(* Logix 5000 project; controller DIMTER vendor 1 type 14 code 77 rev 15.4; software revision 15.01; part 2 of 4 *)
(* tags used below, declared in another part *)
   F : BOOL[2016];   // Flags
   T : TIMER[100];   // Timers
   A123 : ALIAS FOR Local:4:O.Data.3;   // O:4.0/3 A12.3 Reset Buffer
   A142 : ALIAS FOR Local:5:O.Data.2;   // O:5.0/2 A142 Raise Rake 1
   A143 : ALIAS FOR Local:5:O.Data.3;   // O:5.0/3 A143 Brake Cross Conveyor Front of Saw 1
   A144 : ALIAS FOR Local:5:O.Data.4;   // O:5.0/4 A144 Cross Feed 1 Fast Fwd
   A145 : ALIAS FOR Local:5:O.Data.5;   // O:5.0/5 A145 Cross Feed 1 Slow Fwd
   A146 : ALIAS FOR Local:5:O.Data.6;   // O:5.0/6 A146 Cross Feed 1 Fast Rev
   A152 : ALIAS FOR Local:5:O.Data.10;   // O:5.0/10 A15.2 Forward Rotation Rollcase 1
   A156 : ALIAS FOR Local:5:O.Data.14;   // O:5.0/14 A156 Forward Rotation Rollcase 2
   A162 : ALIAS FOR Local:6:O.Data.2;   // O:6.0/2 A16.2 Rake 2
   A163 : ALIAS FOR Local:6:O.Data.3;   // O:6.0/3 A16.3 Brake Cross Conveyor Front of Saw 2
   A164 : ALIAS FOR Local:6:O.Data.4;   // O:6.0/4 A16.4 Cross Feed 2 Fast Fwd
   A165 : ALIAS FOR Local:6:O.Data.5;   // O:6.0/5 A16.5 Cross Feed 2 Slow Fwd
   A166 : ALIAS FOR Local:6:O.Data.6;   // O:6.0/6 A16.6 Cross Feed 2 Fast Rev
   A170 : ALIAS FOR Local:6:O.Data.8;   // O:6.0/8 A17.0 Infeed Measuring Slot Weinig Release Workpiece to Demand
   A171 : ALIAS FOR Local:6:O.Data.9;   // O:6.0/9 A17.1 Conveyor Measuring Slot Weinig Feed to Switch On
   A184 : ALIAS FOR Local:7:O.Data.4;   // O:7.0/4 A18.4 Waste Belt Conveyor 1
   A185 : ALIAS FOR Local:7:O.Data.5;   // O:7.0/5 A18.5 Waste Belt Conveyor 2
   A186 : ALIAS FOR Local:7:O.Data.6;   // O:7.0/6 A18.6 Cross Belt 1
   A187 : ALIAS FOR Local:7:O.Data.7;   // O:7.0/7 A18.7 Cross Belt 2
   E01 : ALIAS FOR Local:1:I.Data.1;   // I:1.0/1 E0.1 Saw Hood 1 Closed
   E02 : ALIAS FOR Local:1:I.Data.2;   // I:1.0/2 E0.2 Saw Motor 1 On
   E05 : ALIAS FOR Local:1:I.Data.5;   // I:1.0/5 E0.5 Failure Chain Ejector
   E06 : ALIAS FOR Local:1:I.Data.6;   // I:1.0/6 E0.6 Failure Conveyor in Front of Saw 1
   E07 : ALIAS FOR Local:1:I.Data.7;   // I:1.0/7 E0.7 Failure Conveyor in Front of Saw 2
   E10 : ALIAS FOR Local:1:I.Data.8;   // I:1.0/8 E1.0 Failure Weinig Conveyor
   E100 : ALIAS FOR Local:3:I.Data.16;   // I:3.1/0 E10.0 Sorting Ejector Sorting 1
   E101 : ALIAS FOR Local:3:I.Data.17;   // I:3.1/1 E10.1 Sorting Ejector 2 Sorting 1
   E102 : ALIAS FOR Local:3:I.Data.18;   // I:3.1/2 E10.2 Sorting Ejector 3 Sorting 1
   E103 : ALIAS FOR Local:3:I.Data.19;   // I:3.1/3 E10.3 Sorting Ejector 1 Sorting 2
   E104 : ALIAS FOR Local:3:I.Data.20;   // I:3.1/4 E10.4 Sorting Ejector 2 Sorting 2
   E105 : ALIAS FOR Local:3:I.Data.21;   // I:3.1/5 E10.5 Sorting Ejector 3 Sorting 2
   E106 : ALIAS FOR Local:3:I.Data.22;   // I:3.1/6 E10.6 Cross Belt 1 Cyclewise Continuous Running
   E107 : ALIAS FOR Local:3:I.Data.23;   // I:3.1/7 E10.7 ???
   E11 : ALIAS FOR Local:1:I.Data.9;   // I:1.0/9 E1.1 Saw Hood 2 Closed
   E110 : ALIAS FOR Local:3:I.Data.24;   // I:3.1/8 E11.0 Cross Belt 1 Footswitch (Removed)
   E111 : ALIAS FOR Local:3:I.Data.25;   // I:3.1/9 E11.1 Cross Belt 2 Cyclewise Continuous Running
   E112 : ALIAS FOR Local:3:I.Data.26;   // I:3.1/10 E11.2 ???
   E113 : ALIAS FOR Local:3:I.Data.27;   // I:3.1/11 E11.3 Cross Belt 2 Footswitch (Removed)
   E114 : ALIAS FOR Local:3:I.Data.28;   // I:3.1/12 E11.4 Transfer Station On
   E115 : ALIAS FOR Local:3:I.Data.29;   // I:3.1/13 E11.5 Cross Feed Manual Fwd-Rev
   E116 : ALIAS FOR Local:3:I.Data.30;   // I:3.1/14 E11.6 ???
   E12 : ALIAS FOR Local:1:I.Data.10;   // I:1.0/10 E1.2 Saw Motor 2 On
   E20 : ALIAS FOR Local:1:I.Data.16;   // I:1.1/0 E2.0 Protection Hood Measuring System
   E27 : ALIAS FOR Local:1:I.Data.23;   // I:1.1/7 E2.7 Reset Safety Barrier at Transfer Station
   E41 : ALIAS FOR Local:2:I.Data.1;   // I:2.0/1 E4.1 Cross Feed 1 Manual Fwd - Rev
   E42 : ALIAS FOR Local:2:I.Data.2;   // I:2.0/2 E4.2 Cross Feed 1 Manual Fwd - Rev
   E44 : ALIAS FOR Local:2:I.Data.4;   // I:2.0/4 E4.4 Waste Conveyor Belt On
   E45 : ALIAS FOR Local:2:I.Data.5;   // I:2.0/5 E4.5 Transfer Station in Front of Saw On
   E51 : ALIAS FOR Local:2:I.Data.9;   // I:2.0/9 E5.1 Cross Feed 2 Manual Fwd - Rev
   E52 : ALIAS FOR Local:2:I.Data.10;   // I:2.0/10 E5.2 Cross Feed 2 Manual Fwd - Rev
   E54 : ALIAS FOR Local:2:I.Data.12;   // I:2.0/12 E5.4 Measuring Station On
   E57 : ALIAS FOR Local:2:I.Data.15;   // I:2.0/15 E5.7 Conveyor Measuring Station Manual
   E67 : ALIAS FOR Local:2:I.Data.23;   // I:2.1/7 E6.7 PE Cross Feed 1 Waiting Position
   E72 : ALIAS FOR Local:2:I.Data.26;   // I:2.1/10 E7.2 Stop Rollcase 1
   E73 : ALIAS FOR Local:2:I.Data.27;   // I:2.1/11 E7.3 Cross Feed 1 Down
   E74 : ALIAS FOR Local:2:I.Data.28;   // I:2.1/12 E7.4 Cross Feed 1 Up
   E75 : ALIAS FOR Local:2:I.Data.29;   // I:2.1/13 E7.5 Cross Feed 1 Initial Position
   E76 : ALIAS FOR Local:2:I.Data.30;   // I:2.1/14 E7.6 PE Cross Feed 1 Slow Fwd
   E77 : ALIAS FOR Local:2:I.Data.31;   // I:2.1/15 E7.7 Cross Feed 1 at Front
   E87 : ALIAS FOR Local:3:I.Data.7;   // I:3.0/7 E8.7 PE Cross Feed 2 Waiting Position
   E92 : ALIAS FOR Local:3:I.Data.10;   // I:3.0/10 E9.2 Stop Rollcase 2
   E93 : ALIAS FOR Local:3:I.Data.11;   // I:3.0/11 E9.3 Cross Feed 2 Down
   E94 : ALIAS FOR Local:3:I.Data.12;   // I:3.0/12 E9.4 Cross Feed 2 Up
   E95 : ALIAS FOR Local:3:I.Data.13;   // I:3.0/13 E9.5 Cross Feed 2 Home Position
   E96 : ALIAS FOR Local:3:I.Data.14;   // I:3.0/14 E9.6 PE Cross Feed 2 Slow Fwd
   E97 : ALIAS FOR Local:3:I.Data.15;   // I:3.0/15 E9.7 Cross Feed 2 at Front
(* MainProgram, continued *)

ROUTINE Conveyors   (* ladder *)
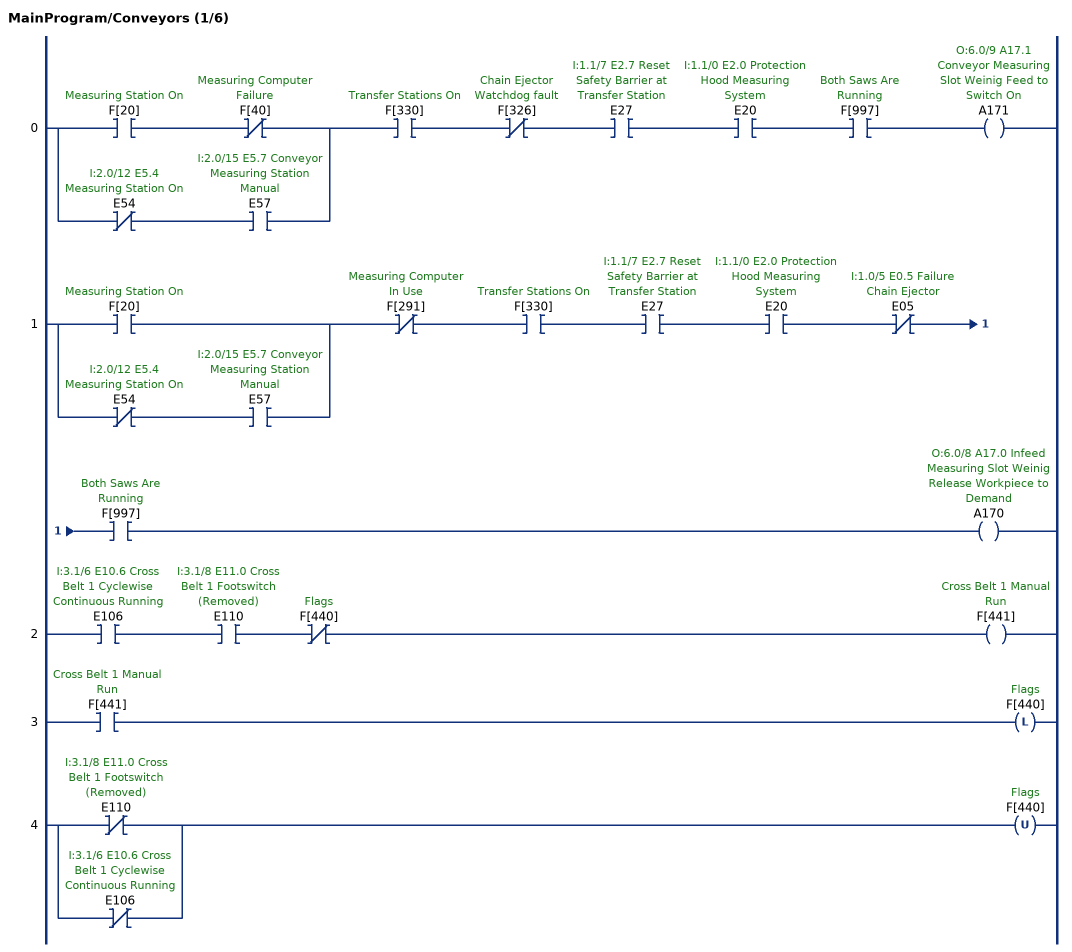
   0: [XIC(F[20]) XIO(F[40]) ,XIO(E54) XIC(E57) ]XIC(F[330])XIO(F[326])XIC(E27)XIC(E20)XIC(F[997])OTE(A171);
   1: [XIC(F[20]) ,XIO(E54) XIC(E57) ]XIO(F[291])XIC(F[330])XIC(E27)XIC(E20)XIO(E05)XIC(F[997])OTE(A170);
   2: XIC(E106)XIC(E110)XIO(F[440])OTE(F[441]);
   3: XIC(F[441])OTL(F[440]);
   4: [XIO(E110) ,XIO(E106) ]OTU(F[440]);
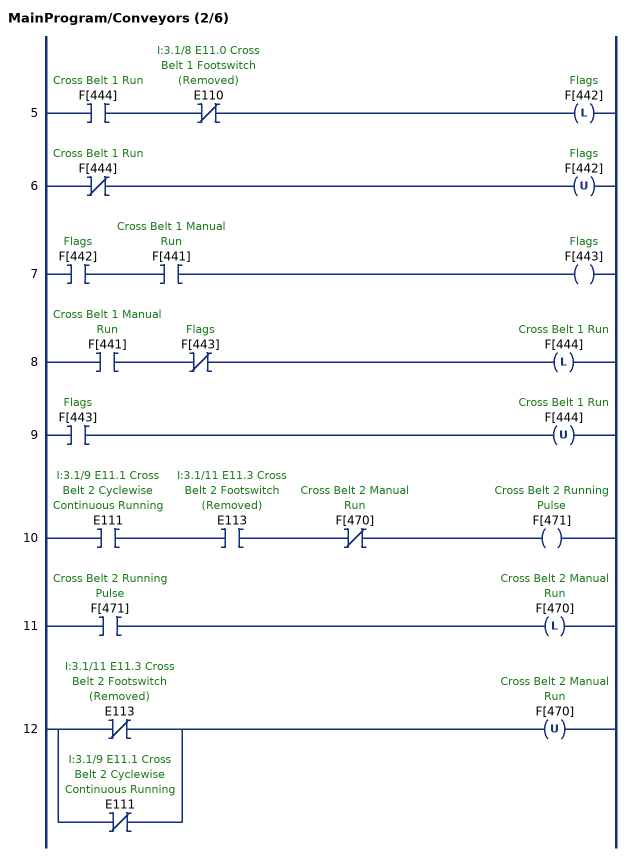
   5: XIC(F[444])XIO(E110)OTL(F[442]);
   6: XIO(F[444])OTU(F[442]);
   7: XIC(F[442])XIC(F[441])OTE(F[443]);
   8: XIC(F[441])XIO(F[443])OTL(F[444]);
   9: XIC(F[443])OTU(F[444]);
   10: XIC(E111)XIC(E113)XIO(F[470])OTE(F[471]);
   11: XIC(F[471])OTL(F[470]);
   12: [XIO(E113) ,XIO(E111) ]OTU(F[470]);
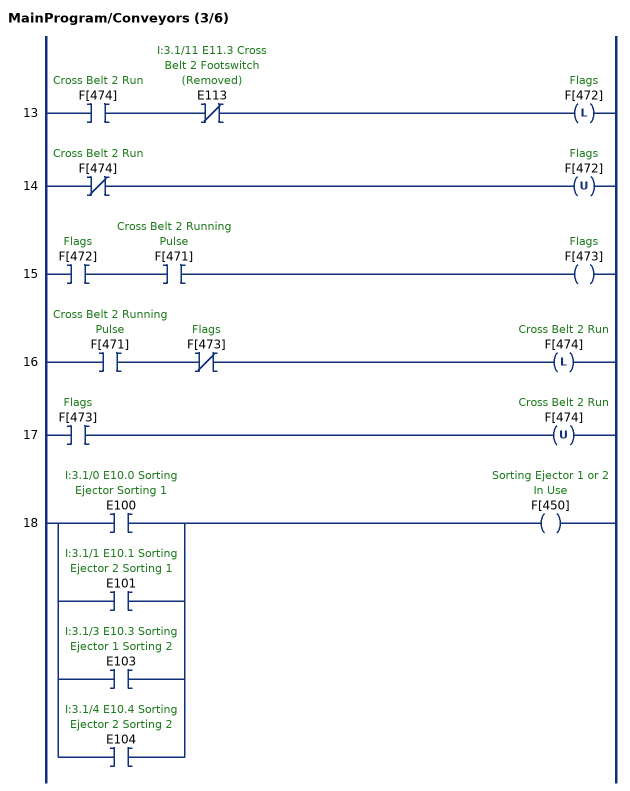
   13: XIC(F[474])XIO(E113)OTL(F[472]);
   14: XIO(F[474])OTU(F[472]);
   15: XIC(F[472])XIC(F[471])OTE(F[473]);
   16: XIC(F[471])XIO(F[473])OTL(F[474]);
   17: XIC(F[473])OTU(F[474]);
   18: [XIC(E100) ,XIC(E101) ,XIC(E103) ,XIC(E104) ]OTE(F[450]);
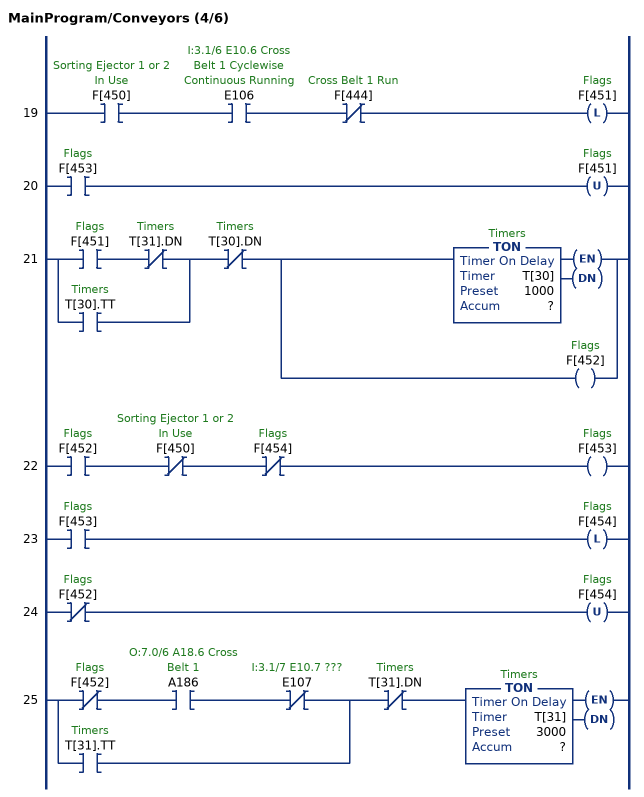
   19: XIC(F[450])XIC(E106)XIO(F[444])OTL(F[451]);
   20: XIC(F[453])OTU(F[451]);
   21: [XIC(F[451]) XIO(T[31].DN) ,XIC(T[30].TT) ]XIO(T[30].DN)[TON(T[30],?,?) ,OTE(F[452]) ];
   22: XIC(F[452])XIO(F[450])XIO(F[454])OTE(F[453]);
   23: XIC(F[453])OTL(F[454]);
   24: XIO(F[452])OTU(F[454]);
   25: [XIO(F[452]) XIC(A186) XIO(E107) ,XIC(T[31].TT) ]XIO(T[31].DN)TON(T[31],?,?);
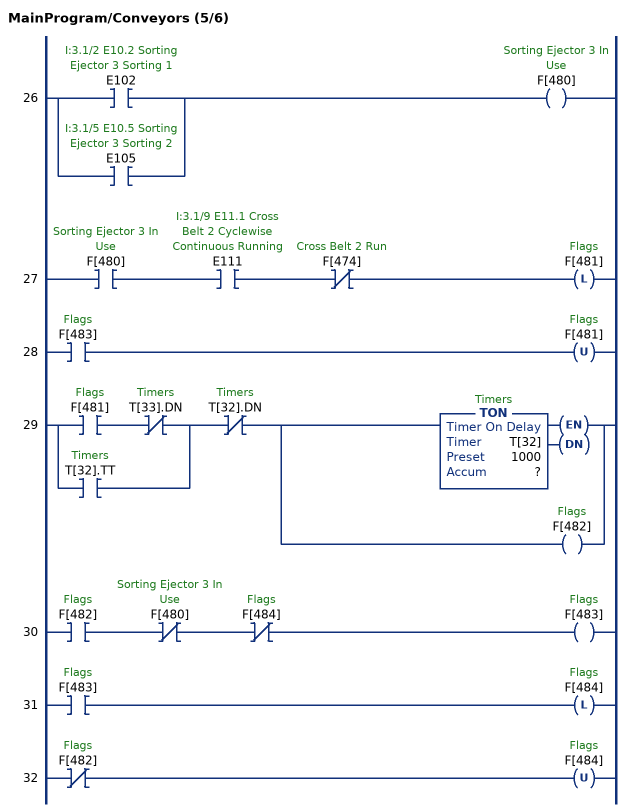
   26: [XIC(E102) ,XIC(E105) ]OTE(F[480]);
   27: XIC(F[480])XIC(E111)XIO(F[474])OTL(F[481]);
   28: XIC(F[483])OTU(F[481]);
   29: [XIC(F[481]) XIO(T[33].DN) ,XIC(T[32].TT) ]XIO(T[32].DN)[TON(T[32],?,?) ,OTE(F[482]) ];
   30: XIC(F[482])XIO(F[480])XIO(F[484])OTE(F[483]);
   31: XIC(F[483])OTL(F[484]);
   32: XIO(F[482])OTU(F[484]);
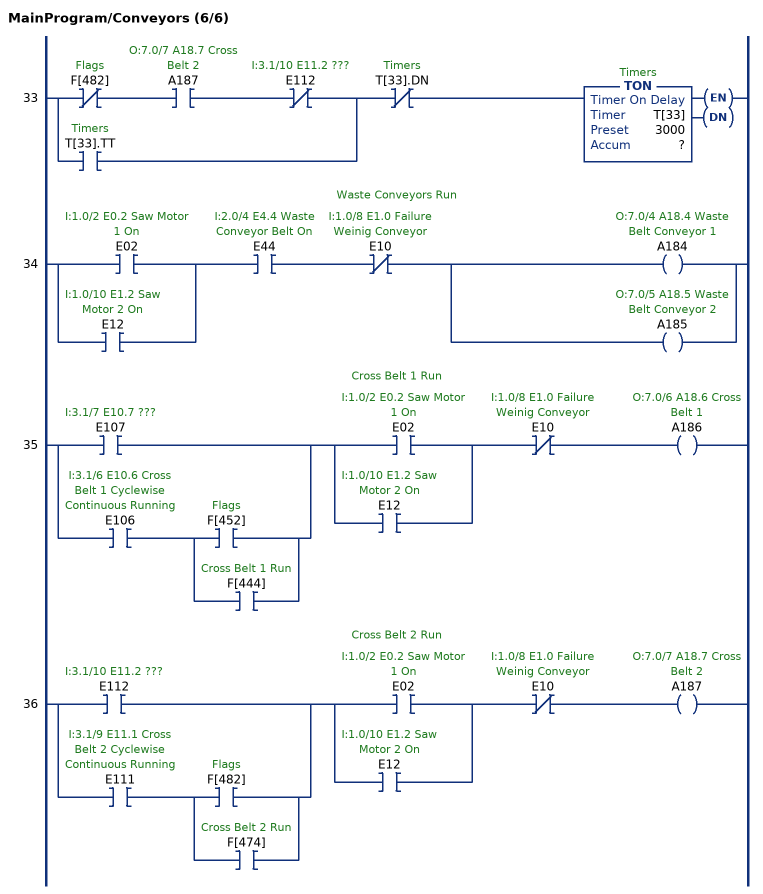
   33: [XIO(F[482]) XIC(A187) XIO(E112) ,XIC(T[33].TT) ]XIO(T[33].DN)TON(T[33],?,?);
   // Waste Conveyors Run
   34: [XIC(E02) ,XIC(E12) ]XIC(E44)XIO(E10)[OTE(A184) ,OTE(A185) ];
   // Cross Belt 1 Run
   35: [XIC(E107) ,XIC(E106) [XIC(F[452]) ,XIC(F[444]) ] ][XIC(E02) ,XIC(E12) ]XIO(E10)OTE(A186);
   // Cross Belt 2 Run
   36: [XIC(E112) ,XIC(E111) [XIC(F[482]) ,XIC(F[474]) ] ][XIC(E02) ,XIC(E12) ]XIO(E10)OTE(A187);
END_ROUTINE

ROUTINE CrossFeeds   (* ladder *)
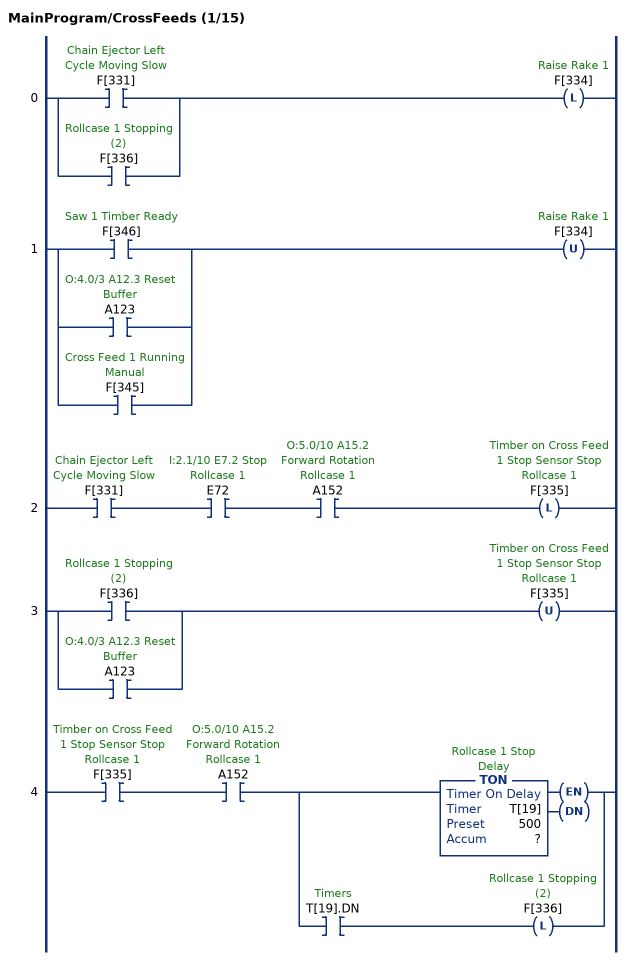
   0: [XIC(F[331]) ,XIC(F[336]) ]OTL(F[334]);
   1: [XIC(F[346]) ,XIC(A123) ,XIC(F[345]) ]OTU(F[334]);
   2: XIC(F[331])XIC(E72)XIC(A152)OTL(F[335]);
   3: [XIC(F[336]) ,XIC(A123) ]OTU(F[335]);
   4: XIC(F[335])XIC(A152)[TON(T[19],?,?) ,XIC(T[19].DN) OTL(F[336]) ];
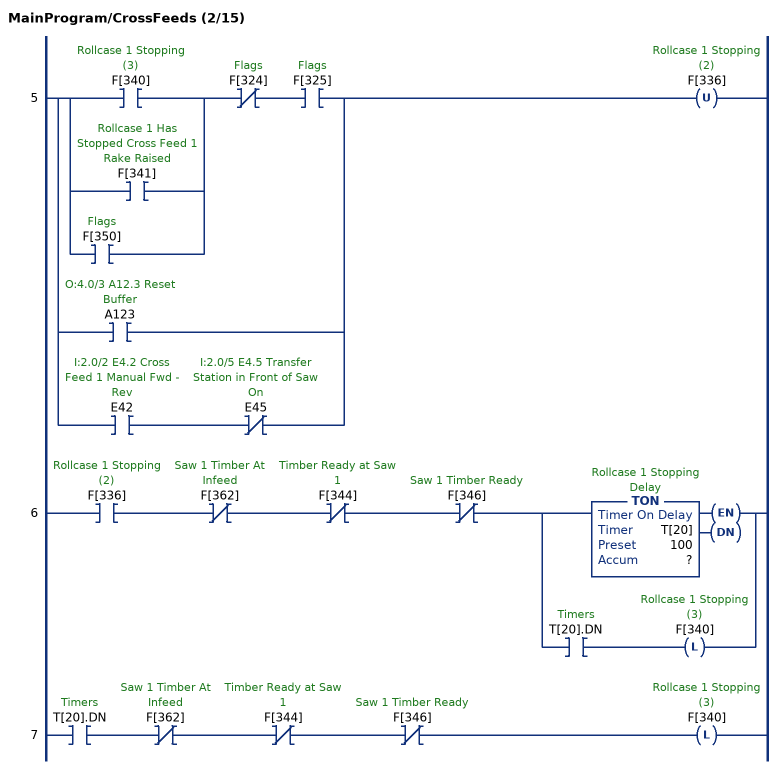
   5: [[XIC(F[340]) ,XIC(F[341]) ,XIC(F[350]) ] XIO(F[324]) XIC(F[325]) ,XIC(A123) ,XIC(E42) XIO(E45) ]OTU(F[336]);
   6: XIC(F[336])XIO(F[362])XIO(F[344])XIO(F[346])[TON(T[20],?,?) ,XIC(T[20].DN) OTL(F[340]) ];
   7: XIC(T[20].DN)XIO(F[362])XIO(F[344])XIO(F[346])OTL(F[340]);
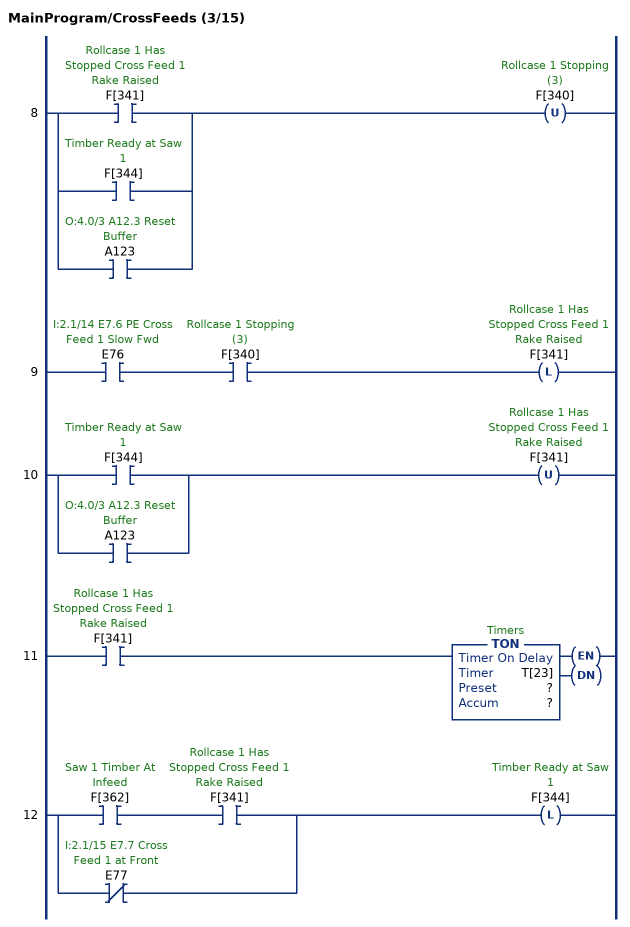
   8: [XIC(F[341]) ,XIC(F[344]) ,XIC(A123) ]OTU(F[340]);
   9: XIC(E76)XIC(F[340])OTL(F[341]);
   10: [XIC(F[344]) ,XIC(A123) ]OTU(F[341]);
   11: XIC(F[341])TON(T[23],?,?);
   12: [XIC(F[362]) XIC(F[341]) ,XIO(E77) ]OTL(F[344]);
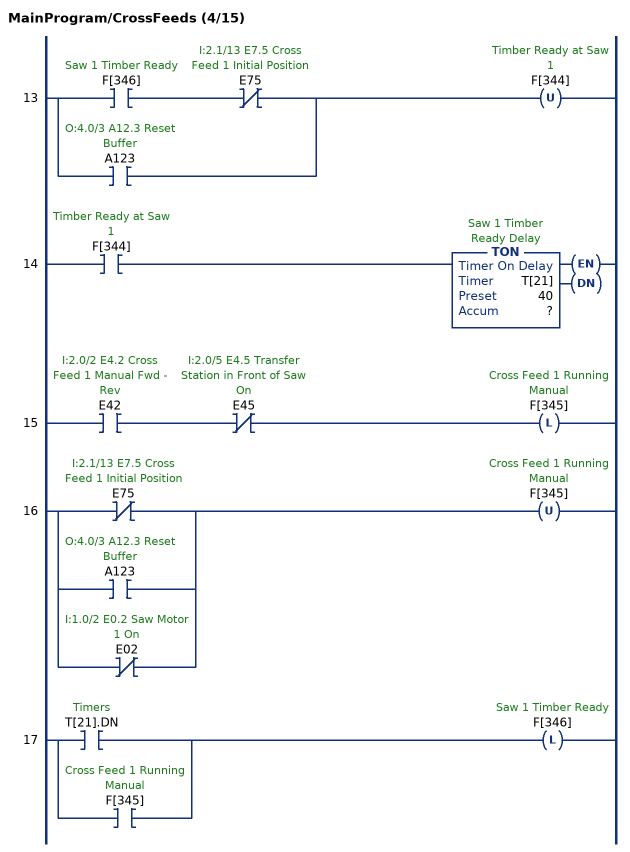
   13: [XIC(F[346]) XIO(E75) ,XIC(A123) ]OTU(F[344]);
   14: XIC(F[344])TON(T[21],?,?);
   15: XIC(E42)XIO(E45)OTL(F[345]);
   16: [XIO(E75) ,XIC(A123) ,XIO(E02) ]OTU(F[345]);
   17: [XIC(T[21].DN) ,XIC(F[345]) ]OTL(F[346]);
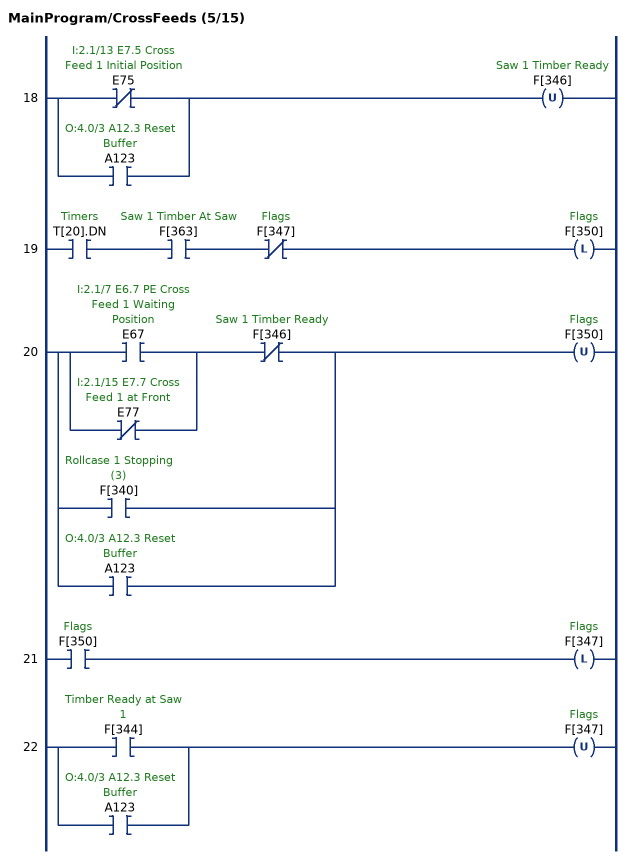
   18: [XIO(E75) ,XIC(A123) ]OTU(F[346]);
   19: XIC(T[20].DN)XIC(F[363])XIO(F[347])OTL(F[350]);
   20: [[XIC(E67) ,XIO(E77) ] XIO(F[346]) ,XIC(F[340]) ,XIC(A123) ]OTU(F[350]);
   21: XIC(F[350])OTL(F[347]);
   22: [XIC(F[344]) ,XIC(A123) ]OTU(F[347]);
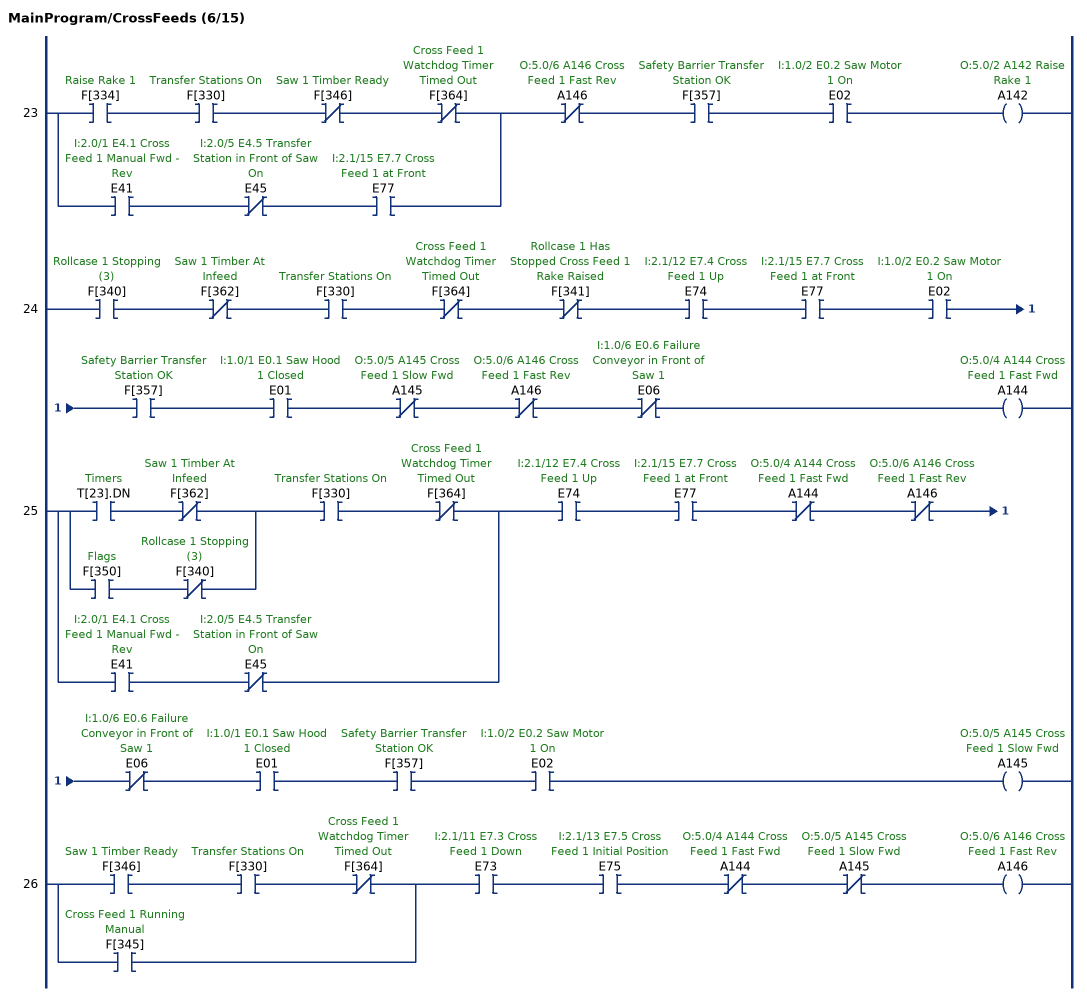
   23: [XIC(F[334]) XIC(F[330]) XIO(F[346]) XIO(F[364]) ,XIC(E41) XIO(E45) XIC(E77) ]XIO(A146)XIC(F[357])XIC(E02)OTE(A142);
   24: XIC(F[340])XIO(F[362])XIC(F[330])XIO(F[364])XIO(F[341])XIC(E74)XIC(E77)XIC(E02)XIC(F[357])XIC(E01)XIO(A145)XIO(A146)XIO(E06)OTE(A144);
   25: [[XIC(T[23].DN) XIO(F[362]) ,XIC(F[350]) XIO(F[340]) ] XIC(F[330]) XIO(F[364]) ,XIC(E41) XIO(E45) ]XIC(E74)XIC(E77)XIO(A144)XIO(A146)XIO(E06)XIC(E01)XIC(F[357])XIC(E02)OTE(A145);
   26: [XIC(F[346]) XIC(F[330]) XIO(F[364]) ,XIC(F[345]) ]XIC(E73)XIC(E75)XIO(A144)XIO(A145)OTE(A146);
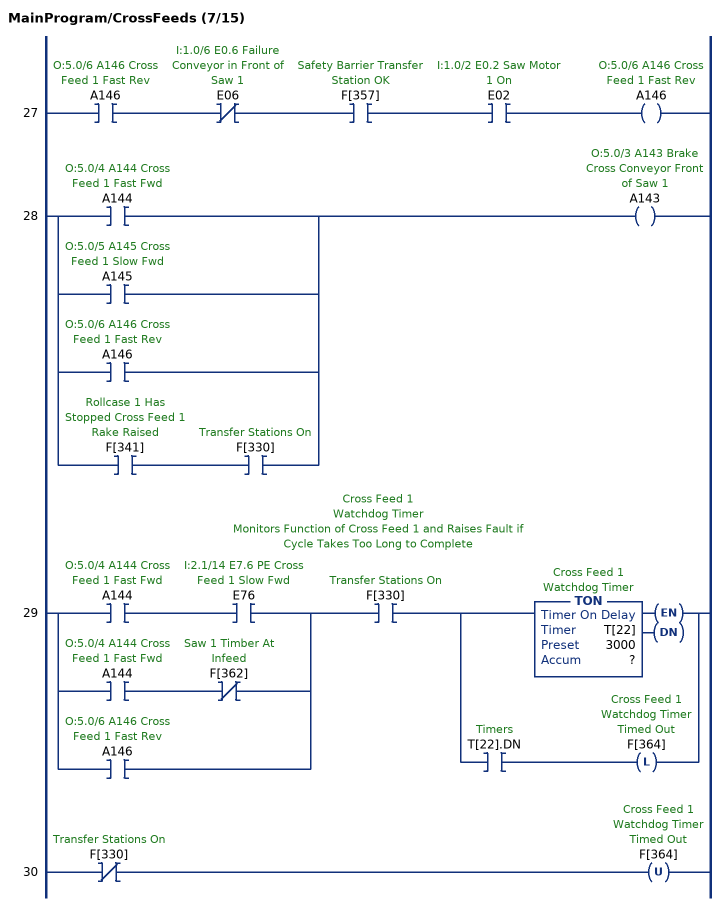
   27: XIC(A146)XIO(E06)XIC(F[357])XIC(E02)OTE(A146);
   28: [XIC(A144) ,XIC(A145) ,XIC(A146) ,XIC(F[341]) XIC(F[330]) ]OTE(A143);
   // Cross Feed 1
   // Watchdog Timer
   // Monitors Function of Cross Feed 1 and Raises Fault if
   // Cycle Takes Too Long to Complete
   29: [XIC(A144) XIC(E76) ,XIC(A144) XIO(F[362]) ,XIC(A146) ]XIC(F[330])[TON(T[22],?,?) ,XIC(T[22].DN) OTL(F[364]) ];
   30: XIO(F[330])OTU(F[364]);
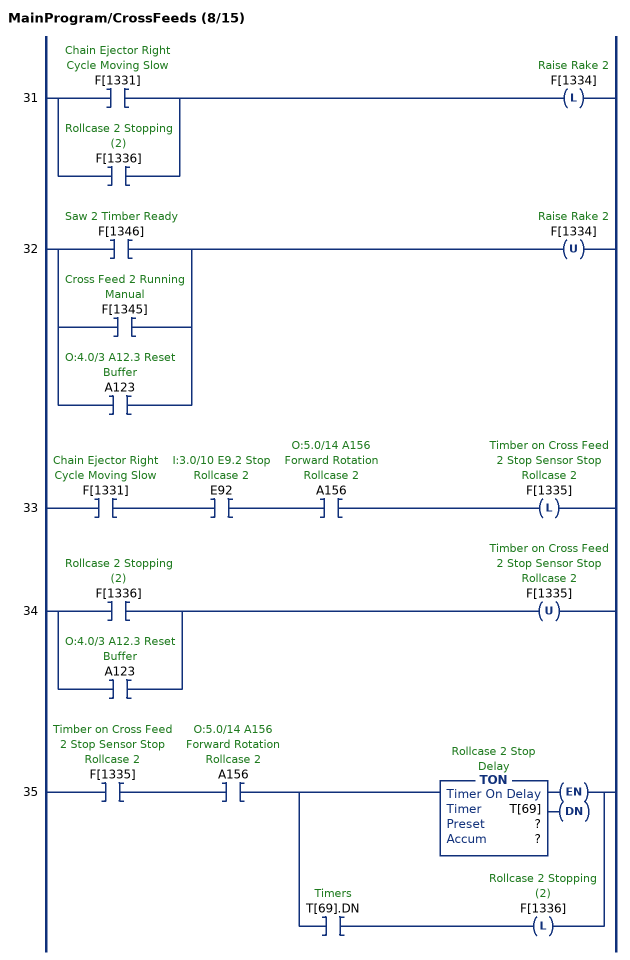
   31: [XIC(F[1331]) ,XIC(F[1336]) ]OTL(F[1334]);
   32: [XIC(F[1346]) ,XIC(F[1345]) ,XIC(A123) ]OTU(F[1334]);
   33: XIC(F[1331])XIC(E92)XIC(A156)OTL(F[1335]);
   34: [XIC(F[1336]) ,XIC(A123) ]OTU(F[1335]);
   35: XIC(F[1335])XIC(A156)[TON(T[69],?,?) ,XIC(T[69].DN) OTL(F[1336]) ];
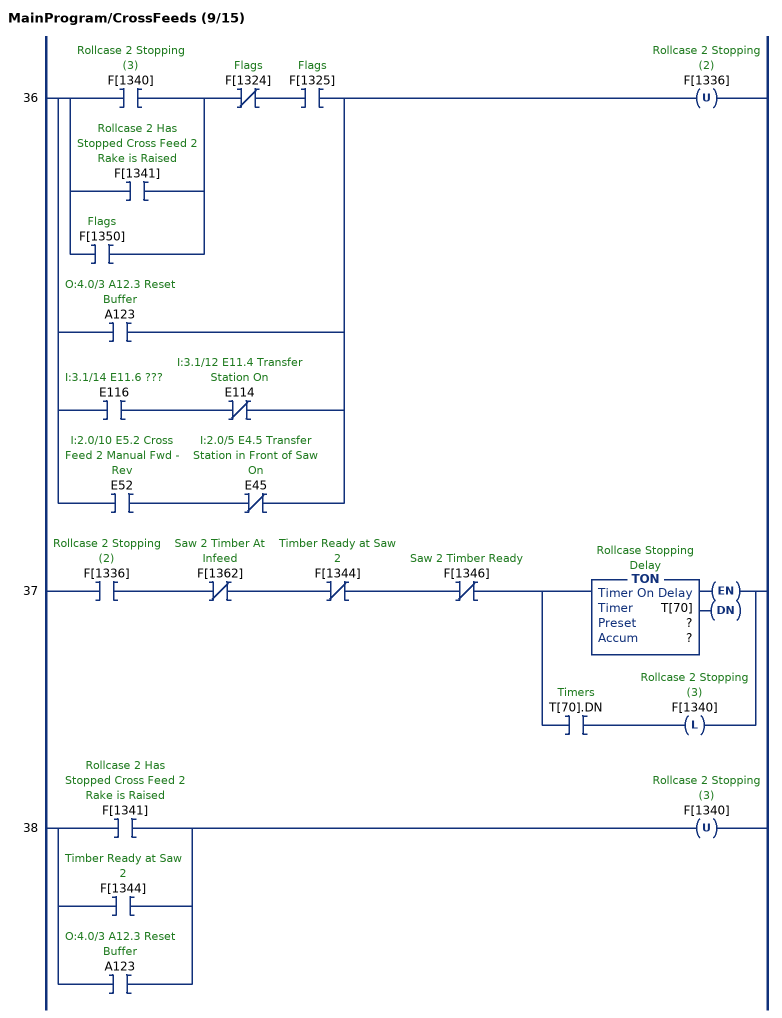
   36: [[XIC(F[1340]) ,XIC(F[1341]) ,XIC(F[1350]) ] XIO(F[1324]) XIC(F[1325]) ,XIC(A123) ,XIC(E116) XIO(E114) ,XIC(E52) XIO(E45) ]OTU(F[1336]);
   37: XIC(F[1336])XIO(F[1362])XIO(F[1344])XIO(F[1346])[TON(T[70],?,?) ,XIC(T[70].DN) OTL(F[1340]) ];
   38: [XIC(F[1341]) ,XIC(F[1344]) ,XIC(A123) ]OTU(F[1340]);
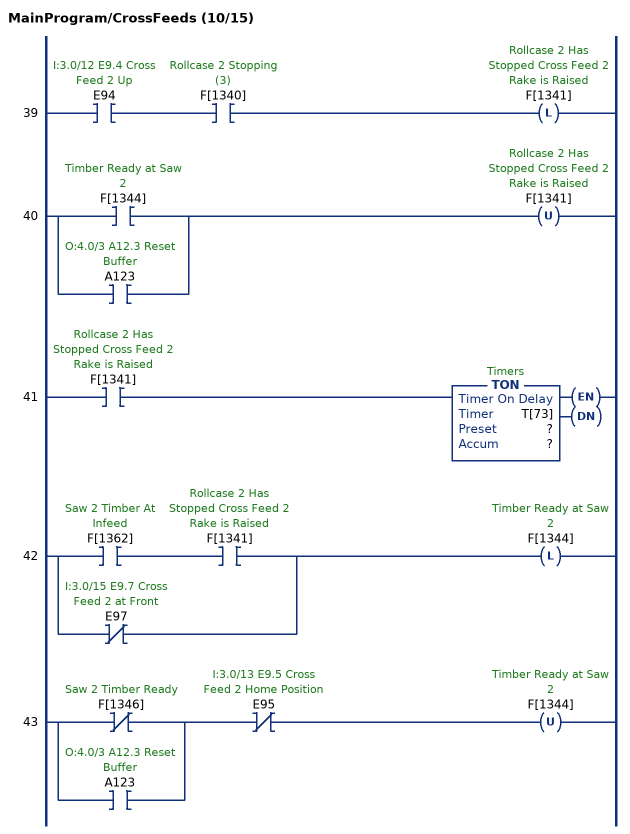
   39: XIC(E94)XIC(F[1340])OTL(F[1341]);
   40: [XIC(F[1344]) ,XIC(A123) ]OTU(F[1341]);
   41: XIC(F[1341])TON(T[73],?,?);
   42: [XIC(F[1362]) XIC(F[1341]) ,XIO(E97) ]OTL(F[1344]);
   43: [XIO(F[1346]) ,XIC(A123) ]XIO(E95)OTU(F[1344]);
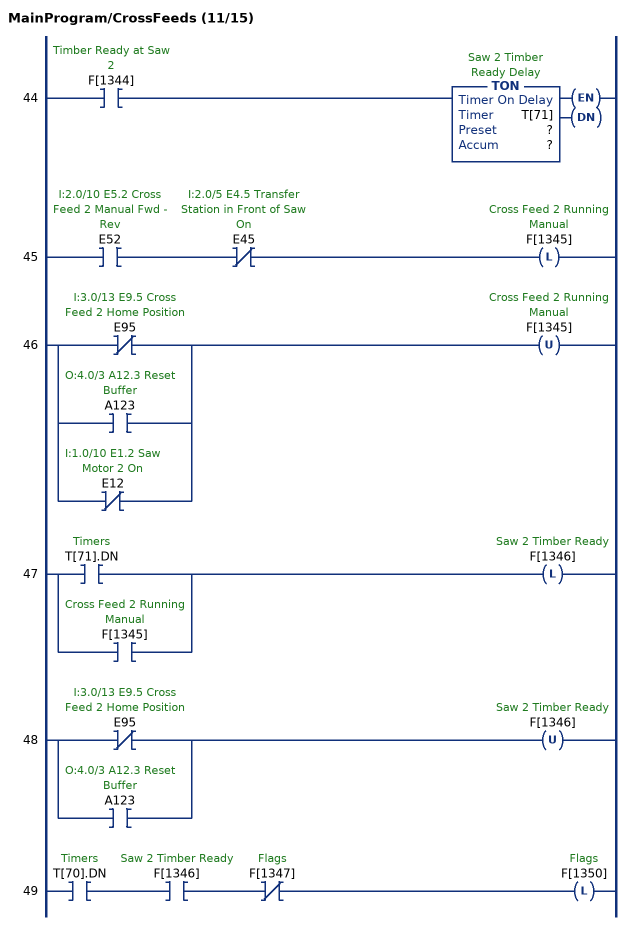
   44: XIC(F[1344])TON(T[71],?,?);
   45: XIC(E52)XIO(E45)OTL(F[1345]);
   46: [XIO(E95) ,XIC(A123) ,XIO(E12) ]OTU(F[1345]);
   47: [XIC(T[71].DN) ,XIC(F[1345]) ]OTL(F[1346]);
   48: [XIO(E95) ,XIC(A123) ]OTU(F[1346]);
   49: XIC(T[70].DN)XIC(F[1346])XIO(F[1347])OTL(F[1350]);
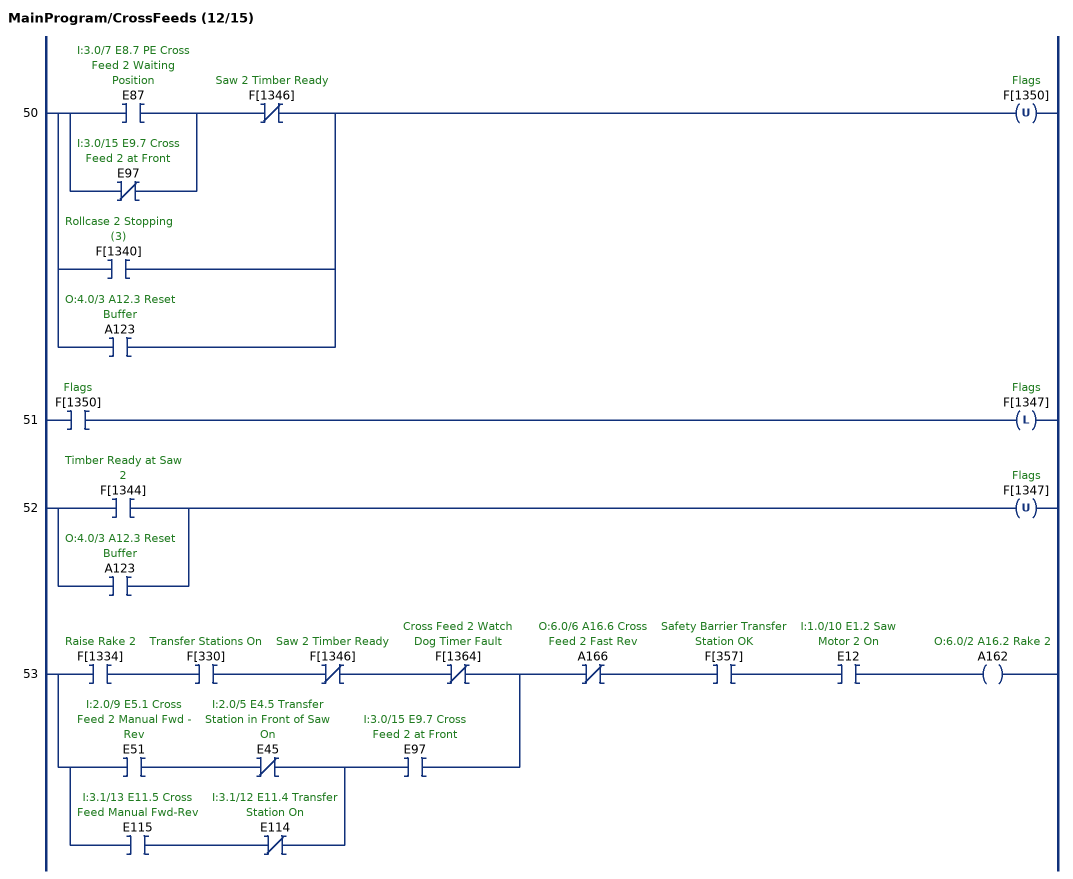
   50: [[XIC(E87) ,XIO(E97) ] XIO(F[1346]) ,XIC(F[1340]) ,XIC(A123) ]OTU(F[1350]);
   51: XIC(F[1350])OTL(F[1347]);
   52: [XIC(F[1344]) ,XIC(A123) ]OTU(F[1347]);
   53: [XIC(F[1334]) XIC(F[330]) XIO(F[1346]) XIO(F[1364]) ,[XIC(E51) XIO(E45) ,XIC(E115) XIO(E114) ] XIC(E97) ]XIO(A166)XIC(F[357])XIC(E12)OTE(A162);
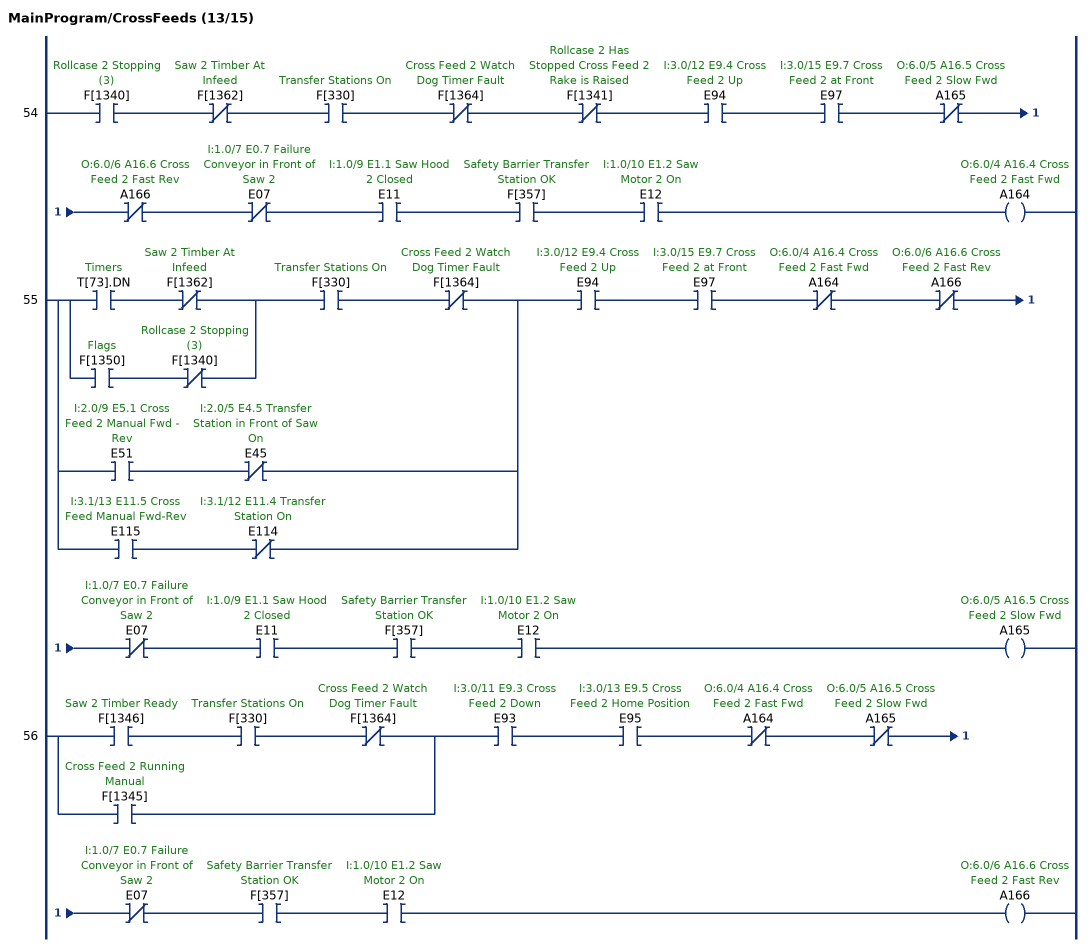
   54: XIC(F[1340])XIO(F[1362])XIC(F[330])XIO(F[1364])XIO(F[1341])XIC(E94)XIC(E97)XIO(A165)XIO(A166)XIO(E07)XIC(E11)XIC(F[357])XIC(E12)OTE(A164);
   55: [[XIC(T[73].DN) XIO(F[1362]) ,XIC(F[1350]) XIO(F[1340]) ] XIC(F[330]) XIO(F[1364]) ,XIC(E51) XIO(E45) ,XIC(E115) XIO(E114) ]XIC(E94)XIC(E97)XIO(A164)XIO(A166)XIO(E07)XIC(E11)XIC(F[357])XIC(E12)OTE(A165);
   56: [XIC(F[1346]) XIC(F[330]) XIO(F[1364]) ,XIC(F[1345]) ]XIC(E93)XIC(E95)XIO(A164)XIO(A165)XIO(E07)XIC(F[357])XIC(E12)OTE(A166);
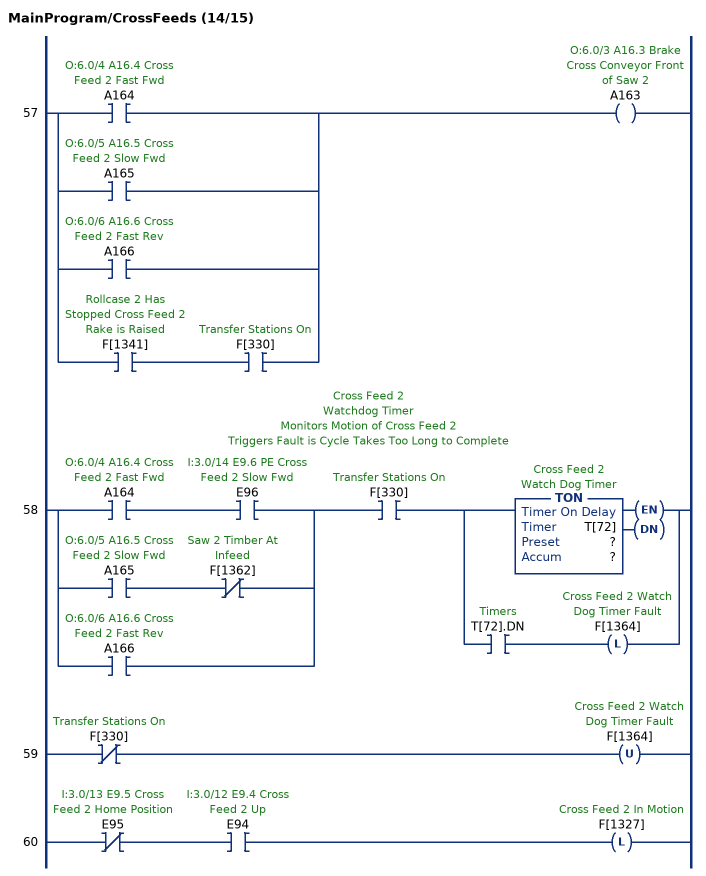
   57: [XIC(A164) ,XIC(A165) ,XIC(A166) ,XIC(F[1341]) XIC(F[330]) ]OTE(A163);
   // Cross Feed 2
   // Watchdog Timer
   // Monitors Motion of Cross Feed 2
   // Triggers Fault is Cycle Takes Too Long to Complete
   58: [XIC(A164) XIC(E96) ,XIC(A165) XIO(F[1362]) ,XIC(A166) ]XIC(F[330])[TON(T[72],?,?) ,XIC(T[72].DN) OTL(F[1364]) ];
   59: XIO(F[330])OTU(F[1364]);
   60: XIO(E95)XIC(E94)OTL(F[1327]);
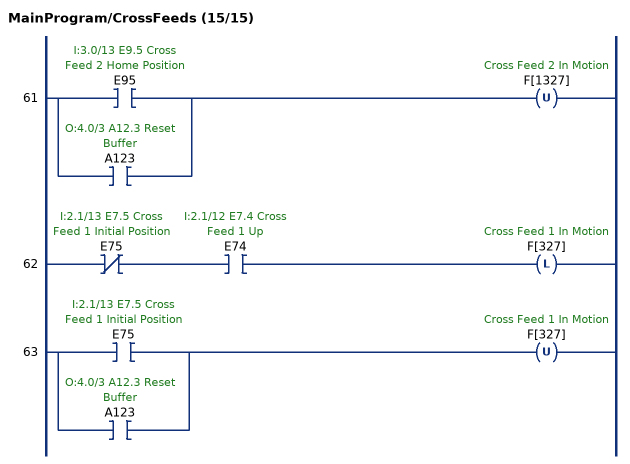
   61: [XIC(E95) ,XIC(A123) ]OTU(F[1327]);
   62: XIO(E75)XIC(E74)OTL(F[327]);
   63: [XIC(E75) ,XIC(A123) ]OTU(F[327]);
END_ROUTINE
